{attribute 'linkalways'} 
{attribute 'no_explicit_call' := 'This FB is a CLASS and must be accessed using methods or properties'}
{attribute 'enable_dynamic_creation'}
FUNCTION_BLOCK _STRING EXTENDS DatatypeBase
VAR
	localData : T_MaxString;
	activeData : REFERENCE TO T_MaxString REF= localData;
END_VAR

PROPERTY PUBLIC Address : PVOID
GET
Address := ADR(activeData);
END_GET
END_PROPERTY

METHOD PUBLIC ClearReference
VAR_INPUT
END_VAR
activeData REF= localData;
END_METHOD

METHOD PUBLIC Clone : I_Datatype
VAR
    pClone : POINTER TO _STRING;
END_VAR
pClone := __NEW(_STRING(InitialValue := Value));
Clone := pClone^;
END_METHOD

METHOD FB_init : BOOL
VAR_INPUT
	bInitRetains : BOOL; // if TRUE, the retain variables are initialized (warm start / cold start)
	bInCopyCode : BOOL;  // if TRUE, the instance afterwards gets moved WORDo the copy code (online change)
	InitialValue : T_MaxString;
END_VAR
localData := InitialValue;
END_METHOD

METHOD PUBLIC MakeReferenceTo
VAR_INPUT
	ReferenceTarget : REFERENCE TO T_MaxString;
END_VAR
activeData REF= ReferenceTarget;
END_METHOD

METHOD PUBLIC SerializeWith
VAR_INPUT
	Serializer : I_Serializer;
END_VAR
Serializer.AddString(activeData);
END_METHOD

PROPERTY PUBLIC Size : UDINT
GET
Size := SIZEOF(activeData);
END_GET
END_PROPERTY

METHOD TryDeserializeFrom : BOOL
VAR_INPUT
	Deserializer : I_Deserializer;
	Feedback : I_DeserializerFeedback;
END_VAR
TryDeserializeFrom := Deserializer.TryGetString(activeData, Feedback);
END_METHOD

METHOD TryMakeReferenceTo : BOOL
VAR_INPUT
	Target : I_Datatype;
END_VAR
VAR
	pTargetData : POINTER TO T_MaxString;
END_VAR
IF NOT (Target.TypeName = TypeName) THEN
	RETURN;
END_IF

pTargetData := Target.Address;
activeData REF= pTargetData^;
TryMakeReferenceTo := TRUE;
END_METHOD

PROPERTY PUBLIC TypeName : T_MAXSTRING
GET
TypeName := 'STRING';
END_GET
END_PROPERTY

PROPERTY PUBLIC Value : REFERENCE TO T_MaxString
GET
Value REF= activeData;
END_GET
END_PROPERTY

END_FUNCTION_BLOCK

(* stored: Version 1.1.0.1, ProductVersion 3.1.4024.12
   POU _STRING: Id {4bcffeea-c7d6-4fdc-9d73-fdf2c3ee34d4}, SpecialFunc None
   Folder Constructor: Id {75dcd086-3f9a-4c88-be97-e59e96f75c99}
   Property Address: Id {cb4bc02b-e0c5-4b50-ab09-b70c3802b828}
   Get Get: Id {e060f5ee-11f2-4fc6-a898-fc18fd9011da}
   Method ClearReference: Id {dc0b0174-64dd-4fda-9700-f7db3b8a081e}
   Method Clone: Id {7bcb1434-bdf5-40a7-a722-535d98637a03}
   Method FB_init: Id {9f96139d-4209-45ef-b1cd-e89dd6ef268f}
   Method MakeReferenceTo: Id {d7e0dade-16b0-4e16-b510-1af01074c622}
   Method SerializeWith: Id {2d3507ad-c5c7-4f71-9b3a-5009da50e599}
   Property Size: Id {63751e4d-e114-4bf8-947b-c543323922db}
   Get Get: Id {3dcdb759-6d97-4be7-883e-684e744456f1}
   Method TryDeserializeFrom: Id {8eb9125c-2dcc-48cd-8370-07590c93daac}
   Method TryMakeReferenceTo: Id {b84d214c-5a47-47c7-b23f-f7eca0db3847}
   Property TypeName: Id {5e31a6dc-b420-4bc2-87df-56fd2777a2bb}
   Get Get: Id {edd11a56-1432-4bcb-8635-abd06eaebc6c}
   Property Value: Id {8be5d6eb-2265-4179-b8c2-35abed67bd8b}
   Get Get: Id {646977de-30b9-4851-be0a-fd6061952fb7} *)
